(* CoDeSys 2.3.9.62 project: WagoAppKNX.SunshadeActuator.pro *)
(* Libraries: C:\Work\WAGO\WAGO.Sandbox\WAGO.KNX\CoDeSys\2.3\DALI_02.lib 27.4.23 19:25:16, C:\Work\WAGO\WAGO.Sandbox\WAGO.KNX\CoDeSys\2.3\KNX_Standard.lib 27.4.23 19:25:16, SysLibGetAddress.lib 7.9.10 15:37:47, C:\Work\WAGO\WAGO.Sandbox\WAGO.KNX\CoDeSys\2.3\mod_com.lib, C:\Work\WAGO\WAGO.Sandbox\WAGO.KNX\CoDeSys\2.3\KNX_Applikations_02.lib 27.4.23 19:25:16, SysLibSockets.lib 16.5.13 14:00:50, NETVARUDP_LIB_V23.LIB*8.11.10 12:37:48, Standard.lib, SYSLIBCALLBACK.LIB, WAGOLibKNXDevice.lib 23.1.08 13:40:44, C:\Work\WAGO\WAGO.Sandbox\WAGO.KNX\CoDeSys\2.3\KNX_IP_750_849_01.lib 27.4.23 19:26:45 *)

(* PLC configuration (modules and I/O channels)
DI_24_0 AT %IX24.0 [BOOLOnX_I] Ch_1 Digital input
AT %IX24.1 [BOOLOnX_I] Ch_2 Digital input
AT %IX24.2 [BOOLOnX_I] Ch_3 Digital input
AT %IX24.3 [BOOLOnX_I] Ch_4 Digital input
AT %IX24.4 [BOOLOnX_I] Ch_5 Digital input
AT %IX24.5 [BOOLOnX_I] Ch_6 Digital input
AT %IX24.6 [BOOLOnX_I] Ch_7 Digital input
AT %IX24.7 [BOOLOnX_I] Ch_8 Digital input
AT %IX24.8 [BOOLOnX_I] Ch_9 Digital input
AT %IX24.9 [BOOLOnX_I] Ch_10 Digital input
AT %IX24.10 [BOOLOnX_I] Ch_11 Digital input
AT %IX24.11 [BOOLOnX_I] Ch_12 Digital input
AT %IX24.12 [BOOLOnX_I] Ch_13 Digital input
AT %IX24.13 [BOOLOnX_I] Ch_14 Digital input
AT %IX24.14 [BOOLOnX_I] Ch_15 Digital input
AT %IX24.15 [BOOLOnX_I] Ch_16 Digital input
AT %IX25.0 [BOOLOnX_I] Ch_1 Digital input
AT %IX25.1 [BOOLOnX_I] Ch_2 Digital input
AT %IX25.2 [BOOLOnX_I] Ch_3 Digital input
AT %IX25.3 [BOOLOnX_I] Ch_4 Digital input
AT %IX25.4 [BOOLOnX_I] Ch_5 Digital input
AT %IX25.5 [BOOLOnX_I] Ch_6 Digital input
AT %IX25.6 [BOOLOnX_I] Ch_7 Digital input
AT %IX25.7 [BOOLOnX_I] Ch_8 Digital input
AT %IX25.8 [BOOLOnX_I] Ch_9 Digital input
AT %IX25.9 [BOOLOnX_I] Ch_10 Digital input
AT %IX25.10 [BOOLOnX_I] Ch_11 Digital input
AT %IX25.11 [BOOLOnX_I] Ch_12 Digital input
AT %IX25.12 [BOOLOnX_I] Ch_13 Digital input
AT %IX25.13 [BOOLOnX_I] Ch_14 Digital input
AT %IX25.14 [BOOLOnX_I] Ch_15 Digital input
AT %IX25.15 [BOOLOnX_I] Ch_16 Digital input
AT %IX26.0 [BOOLOnX_I] Ch_1 Digital input
AT %IX26.1 [BOOLOnX_I] Ch_2 Digital input
AT %IX26.2 [BOOLOnX_I] Ch_3 Digital input
AT %IX26.3 [BOOLOnX_I] Ch_4 Digital input
AT %IX26.4 [BOOLOnX_I] Ch_5 Digital input
AT %IX26.5 [BOOLOnX_I] Ch_6 Digital input
AT %IX26.6 [BOOLOnX_I] Ch_7 Digital input
AT %IX26.7 [BOOLOnX_I] Ch_8 Digital input
AT %IX26.8 [BOOLOnX_I] Ch_9 Digital input
AT %IX26.9 [BOOLOnX_I] Ch_10 Digital input
AT %IX26.10 [BOOLOnX_I] Ch_11 Digital input
AT %IX26.11 [BOOLOnX_I] Ch_12 Digital input
AT %IX26.12 [BOOLOnX_I] Ch_13 Digital input
AT %IX26.13 [BOOLOnX_I] Ch_14 Digital input
AT %IX26.14 [BOOLOnX_I] Ch_15 Digital input
AT %IX26.15 [BOOLOnX_I] Ch_16 Digital input
AT %IX27.0 [BOOLOnX_I] Ch_1 Digital input
AT %IX27.1 [BOOLOnX_I] Ch_2 Digital input
AT %IX27.2 [BOOLOnX_I] Ch_3 Digital input
AT %IX27.3 [BOOLOnX_I] Ch_4 Digital input
AT %IX27.4 [BOOLOnX_I] Ch_5 Digital input
AT %IX27.5 [BOOLOnX_I] Ch_6 Digital input
AT %IX27.6 [BOOLOnX_I] Ch_7 Digital input
AT %IX27.7 [BOOLOnX_I] Ch_8 Digital input
AT %IX27.8 [BOOLOnX_I] Ch_1 Digital input
AT %IX27.9 [BOOLOnX_I] Ch_2 Digital input
AT %IX27.10 [BOOLOnX_I] Ch_3 Digital input
AT %IX27.11 [BOOLOnX_I] Ch_4 Digital input
AT %IX27.12 [BOOLOnX_I] Ch_5 Digital input
AT %IX27.13 [BOOLOnX_I] Ch_6 Digital input
AT %IX27.14 [BOOLOnX_I] Ch_7 Digital input
AT %IX27.15 [BOOLOnX_I] Ch_8 Digital input
DO_24_0 AT %QX24.0 [BOOLOnX_Q] Ch_1 Digital output
AT %QX24.1 [BOOLOnX_Q] Ch_2 Digital output
AT %QX24.2 [BOOLOnX_Q] Ch_3 Digital output
AT %QX24.3 [BOOLOnX_Q] Ch_4 Digital output
AT %QX24.4 [BOOLOnX_Q] Ch_5 Digital output
AT %QX24.5 [BOOLOnX_Q] Ch_6 Digital output
AT %QX24.6 [BOOLOnX_Q] Ch_7 Digital output
AT %QX24.7 [BOOLOnX_Q] Ch_8 Digital output
AT %QX24.8 [BOOLOnX_Q] Ch_9 Digital output
AT %QX24.9 [BOOLOnX_Q] Ch_10 Digital output
AT %QX24.10 [BOOLOnX_Q] Ch_11 Digital output
AT %QX24.11 [BOOLOnX_Q] Ch_12 Digital output
AT %QX24.12 [BOOLOnX_Q] Ch_13 Digital output
AT %QX24.13 [BOOLOnX_Q] Ch_14 Digital output
AT %QX24.14 [BOOLOnX_Q] Ch_15 Digital output
AT %QX24.15 [BOOLOnX_Q] Ch_16 Digital output
0750-1504 16 DO 24V DC 0.5A [Type_10_16_Channels] node 6, in %IB56 out %QB48
  AT %QX25.0 [BOOLOnX_Q] Ch_1 Digital output
  AT %QX25.1 [BOOLOnX_Q] Ch_2 Digital output
  AT %QX25.2 [BOOLOnX_Q] Ch_3 Digital output
  AT %QX25.3 [BOOLOnX_Q] Ch_4 Digital output
  AT %QX25.4 [BOOLOnX_Q] Ch_5 Digital output
  AT %QX25.5 [BOOLOnX_Q] Ch_6 Digital output
  AT %QX25.6 [BOOLOnX_Q] Ch_7 Digital output
  AT %QX25.7 [BOOLOnX_Q] Ch_8 Digital output
  AT %QX25.8 [BOOLOnX_Q] Ch_9 Digital output
  AT %QX25.9 [BOOLOnX_Q] Ch_10 Digital output
  AT %QX25.10 [BOOLOnX_Q] Ch_11 Digital output
  AT %QX25.11 [BOOLOnX_Q] Ch_12 Digital output
  AT %QX25.12 [BOOLOnX_Q] Ch_13 Digital output
  AT %QX25.13 [BOOLOnX_Q] Ch_14 Digital output
  AT %QX25.14 [BOOLOnX_Q] Ch_15 Digital output
  AT %QX25.15 [BOOLOnX_Q] Ch_16 Digital output
0750-1504 16 DO 24V DC 0.5A [Type_10_16_Channels] node 7, in %IB56 out %QB50
  AT %QX26.0 [BOOLOnX_Q] Ch_1 Digital output
  AT %QX26.1 [BOOLOnX_Q] Ch_2 Digital output
  AT %QX26.2 [BOOLOnX_Q] Ch_3 Digital output
  AT %QX26.3 [BOOLOnX_Q] Ch_4 Digital output
  AT %QX26.4 [BOOLOnX_Q] Ch_5 Digital output
  AT %QX26.5 [BOOLOnX_Q] Ch_6 Digital output
  AT %QX26.6 [BOOLOnX_Q] Ch_7 Digital output
  AT %QX26.7 [BOOLOnX_Q] Ch_8 Digital output
  AT %QX26.8 [BOOLOnX_Q] Ch_9 Digital output
  AT %QX26.9 [BOOLOnX_Q] Ch_10 Digital output
  AT %QX26.10 [BOOLOnX_Q] Ch_11 Digital output
  AT %QX26.11 [BOOLOnX_Q] Ch_12 Digital output
  AT %QX26.12 [BOOLOnX_Q] Ch_13 Digital output
  AT %QX26.13 [BOOLOnX_Q] Ch_14 Digital output
  AT %QX26.14 [BOOLOnX_Q] Ch_15 Digital output
  AT %QX26.15 [BOOLOnX_Q] Ch_16 Digital output
0753-0646 KNX-TP1 [Type_30_1_Channels] node 8, in %IB24 out %QB24
  AT %IB0 [BYTEOnB_I] First Byte of 24
  AT %QB0 [BYTEOnB_Q] First Byte of 24
0753-0647 DALI Multi-Master Module [Type_30_1_Channels] node 9, in %IB24 out %QB24
  AT %IB24 [BYTEOnB_I] First Byte of 24
  AT %QB24 [BYTEOnB_Q] First Byte of 24
Modbus variables [PFC200MODBUS] node 1, in %IB0 out %QB0 {PlcStopBehaviour = 1; FiledbusErrorBehaviour = 1; TcpOperation = 1; TcpPort = 502; TcpTimeout = 600; UdpOperation = 1; UdpPort = 502; RtuOperation = 0; NodeId = 1; ResponseTimeout = 100; Interface = 0; Baud = 115200; StopBits = 1; Parity = 1; FlowCtrl = 0; PhysInterface = 0}
Modbus-Master [MB_MASTER] node 2, in %IB0 out %QB0
*)

(* Global variable list: Networkmanagement implicit Variables UDP *)
VAR_GLOBAL CONSTANT
	USE_NWVARS_UDP : BOOL := FALSE;
	MAX_NetVarItems_UDP	: INT := 0;
	MAX_NetVarPDO_Rx_UDP	: INT := 0;
	MAX_NetVarPDO_Tx_UDP	: INT := 0;
	MAX_NetVarOD_UDP		: INT := 0;
END_VAR
VAR_GLOBAL
	pNetVarItems_UDP		: ARRAY[0..MAX_NetVarItems_UDP] OF NetVarDataItem_UDP;
	pNetVarPDO_Rx_UDP		: ARRAY[0..MAX_NetVarPDO_Rx_UDP] OF NetVarPDO_Rx_UDP;
	pNetVarPDO_Tx_UDP		: ARRAY[0..MAX_NetVarPDO_Tx_UDP] OF NetVarPDO_Tx_UDP;
	pNetVarOD_UDP			: ARRAY[0..MAX_NetVarOD_UDP] OF NetVarSDO_UDP;
	pNetVarPDO_Rx_Diagnosis_UDP : ARRAY[0..MAX_NetVarPDO_Rx_UDP] OF NetVarUDPDiagStruct;
	pNetVarPDO_Tx_Diagnosis_UDP : ARRAY[0..MAX_NetVarPDO_Tx_UDP] OF NetVarUDPDiagStruct;
END_VAR

(* POU PLC_PRG, CFC *)
PROGRAM PLC_PRG
VAR
END_VAR
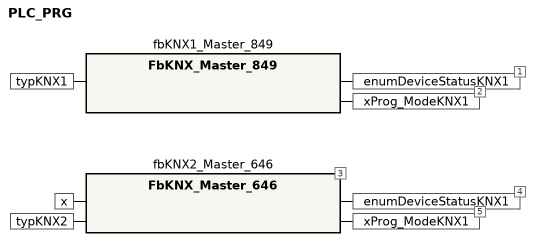
_CFC_ (* Continuous Function Chart, elements in execution order *)
#0 fbKNX1_Master_849:FbKNX_Master_849(typKNX1)
#1 enumDeviceStatusKNX1 <= #0.out 1
#2 xProg_ModeKNX1 <= #0.out 2
#3 fbKNX2_Master_646:FbKNX_Master_646(x, typKNX2)
#4 enumDeviceStatusKNX1 <= #3.out 1
#5 xProg_ModeKNX1 <= #3.out 2
_END_CFC_
END_PROGRAM
